PROGRAM ValveControl
VAR
END_VAR

IF (SEQ.iSeqStepN=0 OR SEQ.iSeqStepN=30) THEN
	VAL.bValve_A_HomeCmd:=TRUE;
	VAL.bValve_A_WorkCmd:=FALSE;
	VAL.bValve_B_HomeCmd:=TRUE;
	VAL.bValve_B_WorkCmd:=FALSE;
	VAL.bValve_C_HomeCmd:=TRUE;
	VAL.bValve_C_WorkCmd:=FALSE;
	VAL.bValve_D_HomeCmd:=TRUE;
	VAL.bValve_D_WorkCmd:=FALSE;
END_IF
//A
IF (SEQ.iSeqStepN=5 OR SEQ.iSeqStepN=10)THEN
	VAL.bValve_A_WorkCmd:=TRUE;
	VAL.bValve_A_HomeCmd :=FALSE;
ELSE
	VAL.bValve_A_WorkCmd:=FALSE;
	VAL.bValve_A_HomeCmd :=TRUE;
END_IF
//B
IF (SEQ.iSeqStepN=10 OR SEQ.iSeqStepN=15)THEN
	VAL.bValve_B_WorkCmd:=TRUE;
	VAL.bValve_B_HomeCmd :=FALSE;
ELSE
	VAL.bValve_B_WorkCmd:=FALSE;
	VAL.bValve_B_HomeCmd :=TRUE;	
END_IF
//C Valve
IF (SEQ.iSeqStepN>=15 AND SEQ.iSeqStepN<=25)THEN
	VAL.bValve_C_WorkCmd:=TRUE;
	VAL.bValve_C_HomeCmd :=FALSE;
ELSE
	VAL.bValve_C_WorkCmd:=FALSE;
	VAL.bValve_C_HomeCmd :=TRUE;	
END_IF

//D Valve
IF (SEQ.iSeqStepN=25)THEN
	VAL.bValve_D_WorkCmd:=TRUE;
	VAL.bValve_D_HomeCmd :=FALSE;
ELSE
	VAL.bValve_D_WorkCmd:=FALSE;
	VAL.bValve_D_HomeCmd :=TRUE;	
END_IF

////Home
//IF (SEQ.iSeqStepN=30)THEN
//	VAL.bValve_D_WorkCmd:=TRUE;
//	VAL.bValve_D_HomeCmd :=FALSE;
//ELSE
//	VAL.bValve_B_WorkCmd:=FALSE;
//	VAL.bValve_B_HomeCmd :=TRUE;	
VAL.bAllValves_At_Home:=VAL.bValve_A_AtHomeSensor AND VAL.bValve_B_AtHomeSensor AND VAL.bValve_C_AtHomeSensor AND VAL.bValve_D_AtHomeSensor;

END_PROGRAM

(* stored: Version 1.1.0.1, ProductVersion 3.1.4024.12
   POU ValveControl: Id {3185a286-a2e9-4973-91ab-229e7cba789e}, SpecialFunc None *)
